Staubli VAL3: remErrArgs.pgx

program remErrArgs(string& sCmd[] (dimensions=1), num& nArgs[] (dimensions=1), num nArgsReq (dimensions=1), string& sReturn[] (dimensions=1))
begin
  // Error raised when we recieve the wrong number of arguments.
  //
  logMsg("call remErrArgs")
  sReturn="ERROR 102"
  sReturn=sReturn+": "+sCmd+" received "
  sReturn=sReturn+toString("",nArgs)
  sReturn=sReturn+" args, expected "
  sReturn=sReturn+toString("",nArgsReq)+"."
  putln(sReturn)
  logMsg(sReturn)
end
